TYPE VALVE :
STRUCT
	jogLeftCmd : BOOL;
	jogRightCmd: BOOL;
	jogValvePos: REAL;
	maxValveMoveRate: REAL;
	velSetpoint: REAL;
	accSetpoint: REAL;
	targetPos: REAL;
	distanceToTarget: REAL;
	moveEnable: BOOL;
	movRight: BOOL;
	movLeft: BOOL;
	autoEnble: BOOL;
	jobEnble: BOOL;
	test: REAL;
END_STRUCT
END_TYPE

(* stored: Version 1.1.0.1
   DUT VALVE: Id {27966e24-a4fd-4cf0-bf0d-d552f9967190} *)
